(* Schneider Machine Expert - Basic project new items, file version 2.0.0.0 *)
(* ProjectInformations: Name=New project *)

HARDWARE
  Cpu 0: TM221CE16R
  EthernetConfiguration: NetworkName=M221, IpAllocationMode=FixedAddress, IpAddress=0.0.0.0, SubnetMask=0.0.0.0
  SerialLineConfiguration: Baud=Baud19200, Parity=ParityEven, DataBits=DataBits8, StopBits=StopBits1, PhysicalMedium=PhysicalMediumRs485, TransmissionMode=TransmissionModeModbusRtu, SlaveId=1, Addressing=SlaveAddressing
  MastTask: UsePeriodScanMode=false, PeriodScan=100
  FastTask: Period=255
  CpuBehavior: StartingMode=StartAsPreviousState, AutoSaveRamOnEeprom=true, WatchdogPeriod=250

SYMBOLS  (address, symbol, comment, settings)
  %SW0      SW_MASTERTASK  "Modifies controller scan period defined at configuration through the user program in the Animation Table Editor"

POU New POU
  (* SectionNumber=1 *)

// Rung 0
  LDR %M10
  [ %MW10 := ROR ( %KW9 , 10 ) ]
  [ %MW1 := ITB ( %KW9 ) ]
  // as ST:
  //   IF RISING(%M10) THEN %MW10 := ROR ( %KW9 , 10 ); END_IF;
  //   IF RISING(%M10) THEN %MW1 := ITB ( %KW9 ); END_IF;

// Rung 1
  LD %M0
  OR %M4
  ST %M2
  // as ST:
  //   %M2 := %M0 OR %M4;

// Rung 2
  LD %M2
  AND( [ %SW0 > %MW0 ]    (* SW_MASTERTASK *)
  OR( %M1
  OPER [ %MW0 := BTI ( %MW10 ) ]
  )
  OR %M5
  )
  ST %M1
  // as ST:
  //   _t1 := SW_MASTERTASK > %MW0;
  //   IF %M1 THEN %MW0 := BTI ( %MW10 ); END_IF;
  //   %M1 := %M2 AND (_t1 OR %M1 OR %M5);
